Yaskawa INFORM job: TEST.JBI

/JOB
//NAME TEST
///FOLDERNAME INNE
//POS
///NPOS 1,1,0,0,0,0
///TOOL 0
///POSTYPE ROBOT
///RECTAN
///RCONF 0,0,0,0,1,0,0,0,0,0,0,0,0,0,0,0,0,0,0,0,0,0,0,0
C00000=236.589,-909.114,-846.591,24.0279,-8.1478,-94.6596
///RCONF 0,0,0,0,0,0,0,0,0,0,0,0,0,0,0,0,0,0,0,0,0,0,0,0
BC00000=1550.023,1886.881,1999.660
//INST
///DATE 2023/11/01 18:40
///ATTR SC,RW,RJ
////FRAME ROBOT
///GROUP1 RB1,BS1
NOP
MOVL C00000 BC00000 V=15.0
END
